# EPICS autosave request: iocBoot/ioc13MeasCompE1608_2/auto_settings.req
file "E1608_settings.req",       P=$(P)
file "pid_control_settings.req"  P=$(P), PID=PID1
